PROGRAM MAIN
VAR
END_VAR

PRG_TXI_VAC();

END_PROGRAM

(* stored: Version 1.1.0.1, ProductVersion 3.1.4024.6
   POU MAIN: Id {e5a9a7ea-bac6-48fa-89f1-5cf69dfbb3cd}, SpecialFunc None *)
